TYPE ST_ActiveEventsHMI :
STRUCT
	sActiveEvents					: T_MaxSTring;
END_STRUCT
END_TYPE

(* stored: Version 1.1.0.1, ProductVersion 3.1.4024.12
   DUT ST_ActiveEventsHMI: Id {19d3e718-4d8c-4ac9-bf1f-d70ec72d6923} *)
